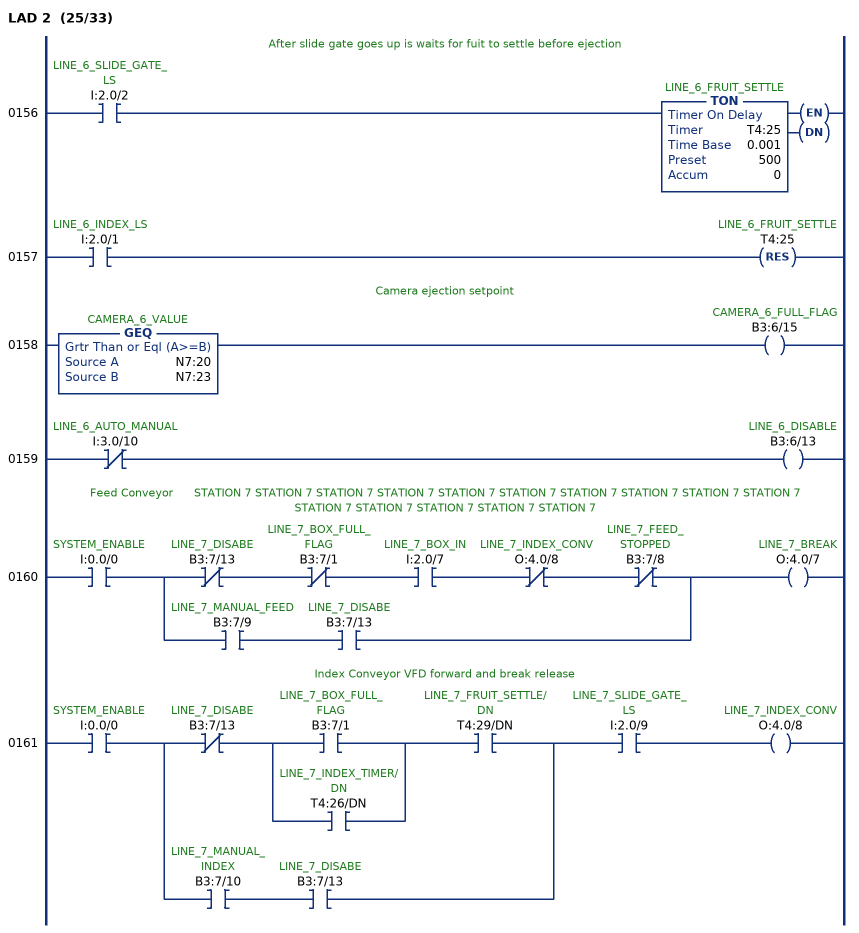
% Rung: 156 %
% After slide gate goes up is waits for fuit to settle before ejection %
SOR XIC I:2.0/2 TON T4:25 0.001 500 0 EOR
%   I:2.0/2  LINE_6_SLIDE_GATE_LS %
%   T4:25  LINE_6_FRUIT_SETTLE %
% Rung: 157 %
SOR XIC I:2.0/1 RES T4:25 EOR
%   I:2.0/1  LINE_6_INDEX_LS %
%   T4:25  LINE_6_FRUIT_SETTLE %
% Rung: 158 %
% Camera ejection setpoint %
SOR GEQ N7:20 N7:23 OTE B3:6/15 EOR
%   N7:20  CAMERA_6_VALUE %
%   N7:23  CAMERA_6_EJECT %
%   B3:6/15  CAMERA_6_FULL_FLAG %
% Rung: 159 %
SOR XIO I:3.0/10 OTE B3:6/13 EOR
%   I:3.0/10  LINE_6_AUTO_MANUAL %
%   B3:6/13  LINE_6_DISABLE %
% Rung: 160 %
% Feed Conveyor      STATION 7 STATION 7 STATION 7 STATION 7 STATION 7 STATION 7 STATION 7 STATION 7 STATION 7 STATION 7 STATION 7 STATION 7 STATION 7 STATION 7 STATION 7 %
SOR XIC I:0.0/0 BST XIO B3:7/13 XIO B3:7/1 XIC I:2.0/7 XIO O:4.0/8 XIO B3:7/8 NXB XIC B3:7/9 XIC B3:7/13 BND OTE O:4.0/7 EOR
%   I:0.0/0  SYSTEM_ENABLE %
%   B3:7/13  LINE_7_DISABE %
%   B3:7/1  LINE_7_BOX_FULL_FLAG %
%   I:2.0/7  LINE_7_BOX_IN %
%   O:4.0/8  LINE_7_INDEX_CONV %
%   B3:7/8  LINE_7_FEED_STOPPED %
%   B3:7/9  LINE_7_MANUAL_FEED %
%   O:4.0/7  LINE_7_BREAK %
% Rung: 161 %
% Index Conveyor VFD forward and break release %
SOR XIC I:0.0/0 BST XIO B3:7/13 BST XIC B3:7/1 NXB XIC T4:26/DN BND XIC T4:29/DN NXB XIC B3:7/10 XIC B3:7/13 BND XIC I:2.0/9 OTE O:4.0/8 EOR
%   I:0.0/0  SYSTEM_ENABLE %
%   B3:7/13  LINE_7_DISABE %
%   B3:7/1  LINE_7_BOX_FULL_FLAG %
%   T4:26  LINE_7_INDEX_TIMER %
%   T4:29  LINE_7_FRUIT_SETTLE %
%   B3:7/10  LINE_7_MANUAL_INDEX %
%   I:2.0/9  LINE_7_SLIDE_GATE_LS %
%   O:4.0/8  LINE_7_INDEX_CONV %

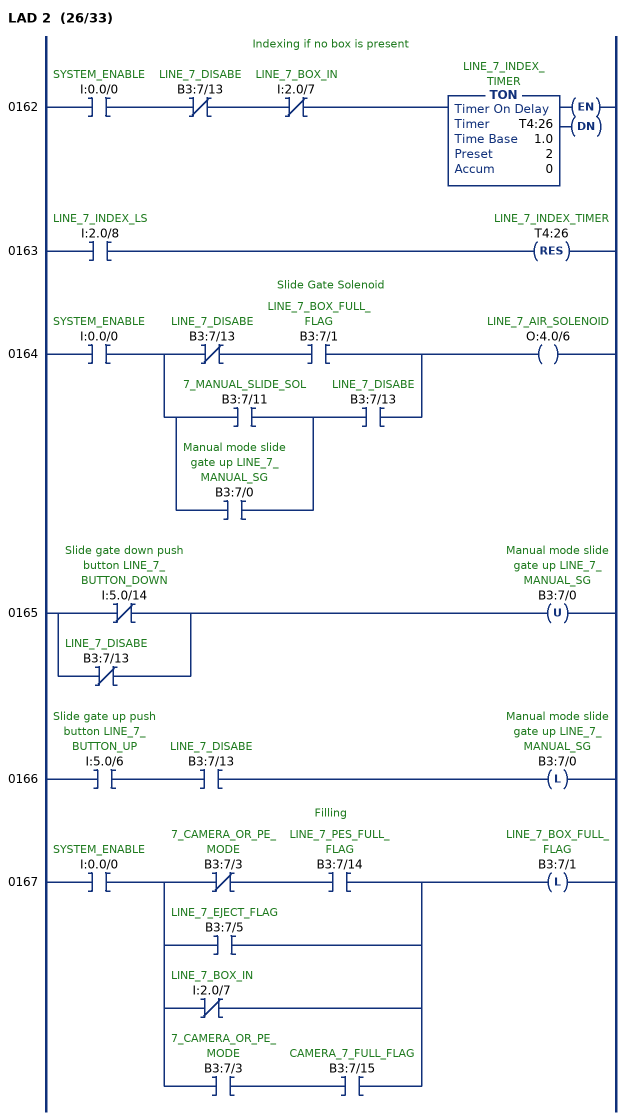
% Rung: 162 %
% Indexing if no box is present %
SOR XIC I:0.0/0 XIO B3:7/13 XIO I:2.0/7 TON T4:26 1.0 2 0 EOR
%   I:0.0/0  SYSTEM_ENABLE %
%   B3:7/13  LINE_7_DISABE %
%   I:2.0/7  LINE_7_BOX_IN %
%   T4:26  LINE_7_INDEX_TIMER %
% Rung: 163 %
SOR XIC I:2.0/8 RES T4:26 EOR
%   I:2.0/8  LINE_7_INDEX_LS %
%   T4:26  LINE_7_INDEX_TIMER %
% Rung: 164 %
% Slide Gate Solenoid %
SOR XIC I:0.0/0 BST XIO B3:7/13 XIC B3:7/1 NXB BST XIC B3:7/11 NXB XIC B3:7/0 BND XIC B3:7/13 BND OTE O:4.0/6 EOR
%   I:0.0/0  SYSTEM_ENABLE %
%   B3:7/13  LINE_7_DISABE %
%   B3:7/1  LINE_7_BOX_FULL_FLAG %
%   B3:7/11  7_MANUAL_SLIDE_SOL %
%   B3:7/0  LINE_7_MANUAL_SG  "Manual mode slide gate up" %
%   O:4.0/6  LINE_7_AIR_SOLENOID %
% Rung: 165 %
SOR BST XIO I:5.0/14 NXB XIO B3:7/13 BND OTU B3:7/0 EOR
%   I:5.0/14  LINE_7_BUTTON_DOWN  "Slide gate down push button" %
%   B3:7/13  LINE_7_DISABE %
%   B3:7/0  LINE_7_MANUAL_SG  "Manual mode slide gate up" %
% Rung: 166 %
SOR XIC I:5.0/6 XIC B3:7/13 OTL B3:7/0 EOR
%   I:5.0/6  LINE_7_BUTTON_UP  "Slide gate up push button" %
%   B3:7/13  LINE_7_DISABE %
%   B3:7/0  LINE_7_MANUAL_SG  "Manual mode slide gate up" %
% Rung: 167 %
% Filling %
SOR XIC I:0.0/0 BST XIO B3:7/3 XIC B3:7/14 NXB BST XIC B3:7/5 NXB BST XIO I:2.0/7 NXB XIC B3:7/3 XIC B3:7/15 BND BND BND OTL B3:7/1 EOR
%   I:0.0/0  SYSTEM_ENABLE %
%   B3:7/3  7_CAMERA_OR_PE_MODE %
%   B3:7/14  LINE_7_PES_FULL_FLAG %
%   B3:7/5  LINE_7_EJECT_FLAG %
%   I:2.0/7  LINE_7_BOX_IN %
%   B3:7/15  CAMERA_7_FULL_FLAG %
%   B3:7/1  LINE_7_BOX_FULL_FLAG %

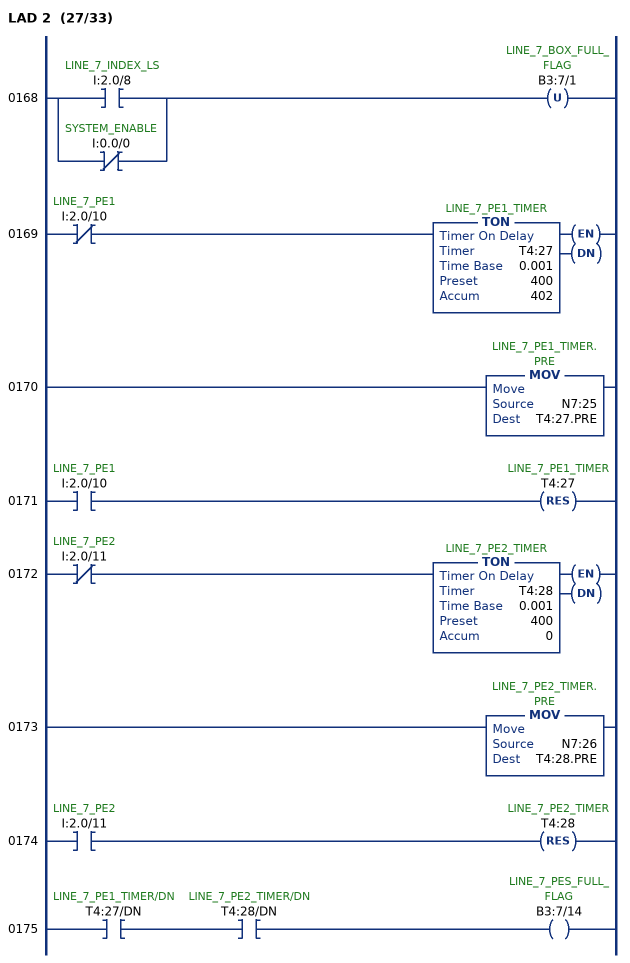
% Rung: 168 %
SOR BST XIC I:2.0/8 NXB XIO I:0.0/0 BND OTU B3:7/1 EOR
%   I:2.0/8  LINE_7_INDEX_LS %
%   I:0.0/0  SYSTEM_ENABLE %
%   B3:7/1  LINE_7_BOX_FULL_FLAG %
% Rung: 169 %
SOR XIO I:2.0/10 TON T4:27 0.001 400 402 EOR
%   I:2.0/10  LINE_7_PE1 %
%   T4:27  LINE_7_PE1_TIMER %
% Rung: 170 %
SOR MOV N7:25 T4:27.PRE EOR
%   N7:25  LINE_7_PE1_TIME_MOV %
%   T4:27  LINE_7_PE1_TIMER %
% Rung: 171 %
SOR XIC I:2.0/10 RES T4:27 EOR
%   I:2.0/10  LINE_7_PE1 %
%   T4:27  LINE_7_PE1_TIMER %
% Rung: 172 %
SOR XIO I:2.0/11 TON T4:28 0.001 400 0 EOR
%   I:2.0/11  LINE_7_PE2 %
%   T4:28  LINE_7_PE2_TIMER %
% Rung: 173 %
SOR MOV N7:26 T4:28.PRE EOR
%   N7:26  LINE_7_PE2_TIME_MOV %
%   T4:28  LINE_7_PE2_TIMER %
% Rung: 174 %
SOR XIC I:2.0/11 RES T4:28 EOR
%   I:2.0/11  LINE_7_PE2 %
%   T4:28  LINE_7_PE2_TIMER %
% Rung: 175 %
SOR XIC T4:27/DN XIC T4:28/DN OTE B3:7/14 EOR
%   T4:27  LINE_7_PE1_TIMER %
%   T4:28  LINE_7_PE2_TIMER %
%   B3:7/14  LINE_7_PES_FULL_FLAG %

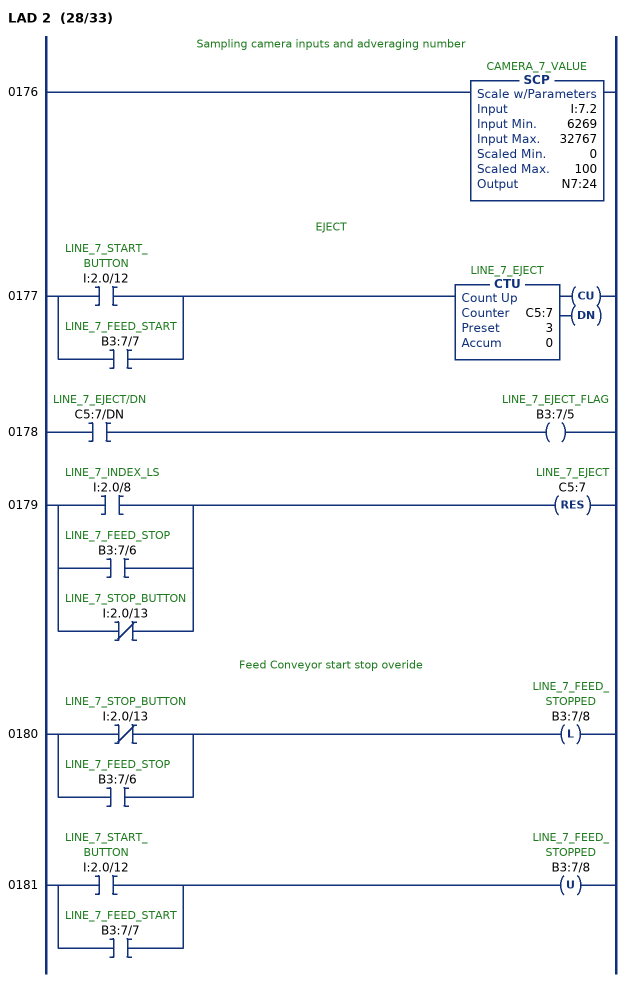
% Rung: 176 %
% Sampling camera inputs and adveraging number %
SOR SCP I:7.2 6269 32767 0 100 N7:24 EOR
%   N7:24  CAMERA_7_VALUE %
% Rung: 177 %
% EJECT %
SOR BST XIC I:2.0/12 NXB XIC B3:7/7 BND CTU C5:7 3 0 EOR
%   I:2.0/12  LINE_7_START_BUTTON %
%   B3:7/7  LINE_7_FEED_START %
%   C5:7  LINE_7_EJECT %
% Rung: 178 %
SOR XIC C5:7/DN OTE B3:7/5 EOR
%   C5:7  LINE_7_EJECT %
%   B3:7/5  LINE_7_EJECT_FLAG %
% Rung: 179 %
SOR BST XIC I:2.0/8 NXB BST XIC B3:7/6 NXB XIO I:2.0/13 BND BND RES C5:7 EOR
%   I:2.0/8  LINE_7_INDEX_LS %
%   B3:7/6  LINE_7_FEED_STOP %
%   I:2.0/13  LINE_7_STOP_BUTTON %
%   C5:7  LINE_7_EJECT %
% Rung: 180 %
% Feed Conveyor start stop overide %
SOR BST XIO I:2.0/13 NXB XIC B3:7/6 BND OTL B3:7/8 EOR
%   I:2.0/13  LINE_7_STOP_BUTTON %
%   B3:7/6  LINE_7_FEED_STOP %
%   B3:7/8  LINE_7_FEED_STOPPED %
% Rung: 181 %
SOR BST XIC I:2.0/12 NXB XIC B3:7/7 BND OTU B3:7/8 EOR
%   I:2.0/12  LINE_7_START_BUTTON %
%   B3:7/7  LINE_7_FEED_START %
%   B3:7/8  LINE_7_FEED_STOPPED %

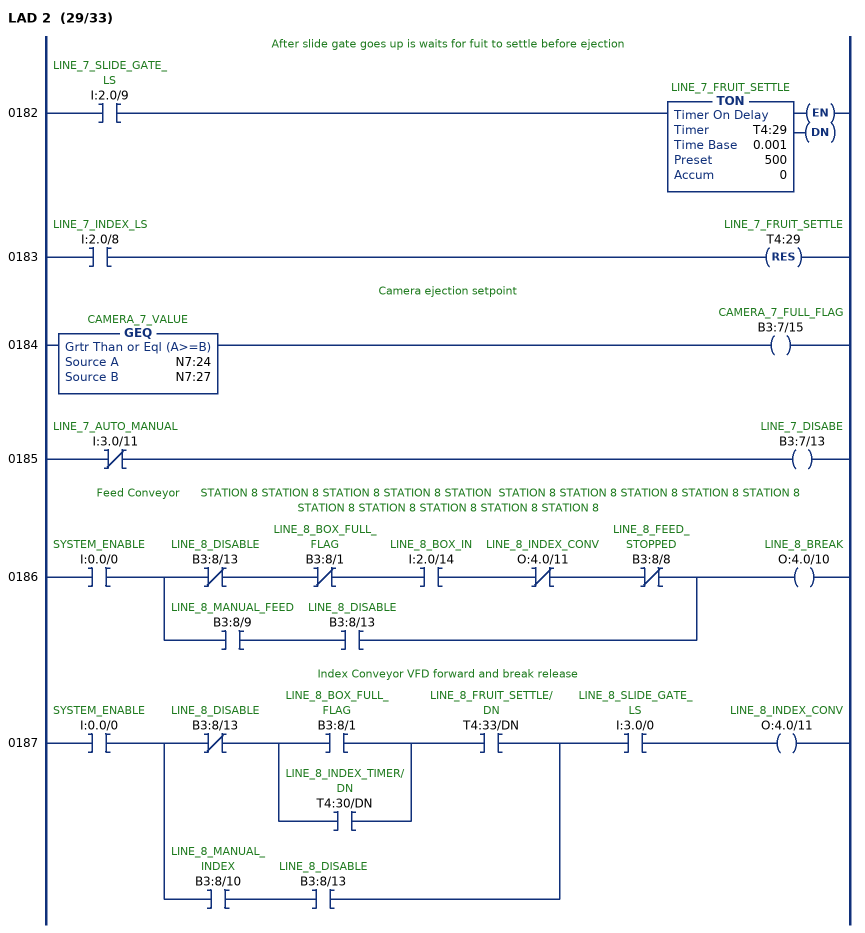
% Rung: 182 %
% After slide gate goes up is waits for fuit to settle before ejection %
SOR XIC I:2.0/9 TON T4:29 0.001 500 0 EOR
%   I:2.0/9  LINE_7_SLIDE_GATE_LS %
%   T4:29  LINE_7_FRUIT_SETTLE %
% Rung: 183 %
SOR XIC I:2.0/8 RES T4:29 EOR
%   I:2.0/8  LINE_7_INDEX_LS %
%   T4:29  LINE_7_FRUIT_SETTLE %
% Rung: 184 %
% Camera ejection setpoint %
SOR GEQ N7:24 N7:27 OTE B3:7/15 EOR
%   N7:24  CAMERA_7_VALUE %
%   N7:27  CAMERA_7_EJECT %
%   B3:7/15  CAMERA_7_FULL_FLAG %
% Rung: 185 %
SOR XIO I:3.0/11 OTE B3:7/13 EOR
%   I:3.0/11  LINE_7_AUTO_MANUAL %
%   B3:7/13  LINE_7_DISABE %
% Rung: 186 %
% Feed Conveyor      STATION 8 STATION 8 STATION 8 STATION 8 STATION  STATION 8 STATION 8 STATION 8 STATION 8 STATION 8 STATION 8 STATION 8 STATION 8 STATION 8 STATION 8 %
SOR XIC I:0.0/0 BST XIO B3:8/13 XIO B3:8/1 XIC I:2.0/14 XIO O:4.0/11 XIO B3:8/8 NXB XIC B3:8/9 XIC B3:8/13 BND OTE O:4.0/10 EOR
%   I:0.0/0  SYSTEM_ENABLE %
%   B3:8/13  LINE_8_DISABLE %
%   B3:8/1  LINE_8_BOX_FULL_FLAG %
%   I:2.0/14  LINE_8_BOX_IN %
%   O:4.0/11  LINE_8_INDEX_CONV %
%   B3:8/8  LINE_8_FEED_STOPPED %
%   B3:8/9  LINE_8_MANUAL_FEED %
%   O:4.0/10  LINE_8_BREAK %
% Rung: 187 %
% Index Conveyor VFD forward and break release %
SOR XIC I:0.0/0 BST XIO B3:8/13 BST XIC B3:8/1 NXB XIC T4:30/DN BND XIC T4:33/DN NXB XIC B3:8/10 XIC B3:8/13 BND XIC I:3.0/0 OTE O:4.0/11 EOR
%   I:0.0/0  SYSTEM_ENABLE %
%   B3:8/13  LINE_8_DISABLE %
%   B3:8/1  LINE_8_BOX_FULL_FLAG %
%   T4:30  LINE_8_INDEX_TIMER %
%   T4:33  LINE_8_FRUIT_SETTLE %
%   B3:8/10  LINE_8_MANUAL_INDEX %
%   I:3.0/0  LINE_8_SLIDE_GATE_LS %
%   O:4.0/11  LINE_8_INDEX_CONV %

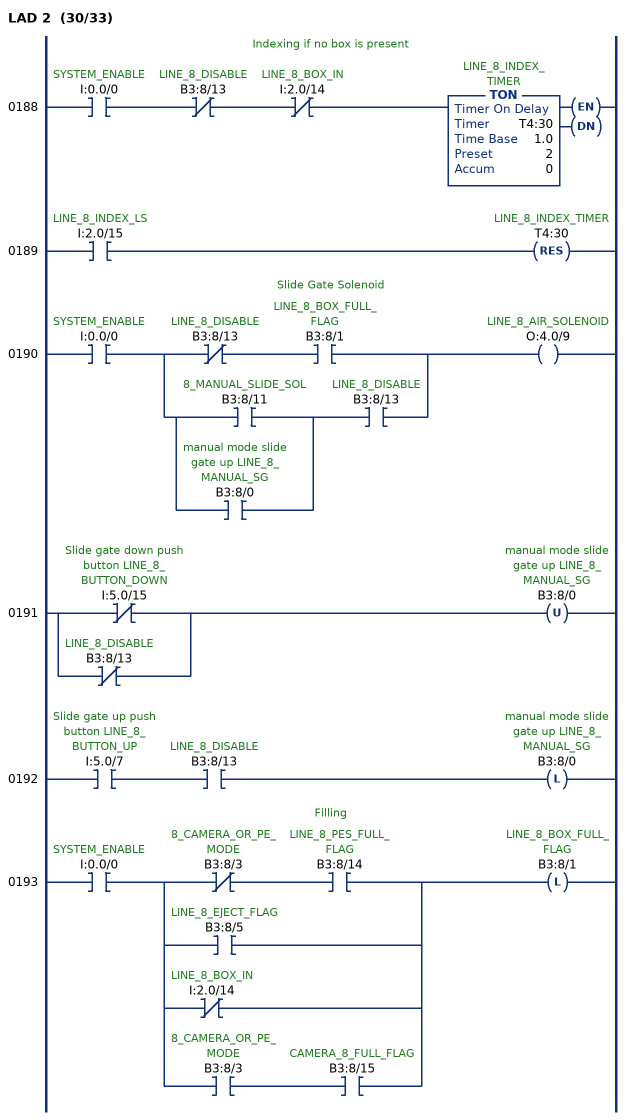
% Rung: 188 %
% Indexing if no box is present %
SOR XIC I:0.0/0 XIO B3:8/13 XIO I:2.0/14 TON T4:30 1.0 2 0 EOR
%   I:0.0/0  SYSTEM_ENABLE %
%   B3:8/13  LINE_8_DISABLE %
%   I:2.0/14  LINE_8_BOX_IN %
%   T4:30  LINE_8_INDEX_TIMER %
% Rung: 189 %
SOR XIC I:2.0/15 RES T4:30 EOR
%   I:2.0/15  LINE_8_INDEX_LS %
%   T4:30  LINE_8_INDEX_TIMER %
% Rung: 190 %
% Slide Gate Solenoid %
SOR XIC I:0.0/0 BST XIO B3:8/13 XIC B3:8/1 NXB BST XIC B3:8/11 NXB XIC B3:8/0 BND XIC B3:8/13 BND OTE O:4.0/9 EOR
%   I:0.0/0  SYSTEM_ENABLE %
%   B3:8/13  LINE_8_DISABLE %
%   B3:8/1  LINE_8_BOX_FULL_FLAG %
%   B3:8/11  8_MANUAL_SLIDE_SOL %
%   B3:8/0  LINE_8_MANUAL_SG  "manual mode slide gate up" %
%   O:4.0/9  LINE_8_AIR_SOLENOID %
% Rung: 191 %
SOR BST XIO I:5.0/15 NXB XIO B3:8/13 BND OTU B3:8/0 EOR
%   I:5.0/15  LINE_8_BUTTON_DOWN  "Slide gate down push button" %
%   B3:8/13  LINE_8_DISABLE %
%   B3:8/0  LINE_8_MANUAL_SG  "manual mode slide gate up" %
% Rung: 192 %
SOR XIC I:5.0/7 XIC B3:8/13 OTL B3:8/0 EOR
%   I:5.0/7  LINE_8_BUTTON_UP  "Slide gate up push button" %
%   B3:8/13  LINE_8_DISABLE %
%   B3:8/0  LINE_8_MANUAL_SG  "manual mode slide gate up" %
% Rung: 193 %
% Filling %
SOR XIC I:0.0/0 BST XIO B3:8/3 XIC B3:8/14 NXB BST XIC B3:8/5 NXB BST XIO I:2.0/14 NXB XIC B3:8/3 XIC B3:8/15 BND BND BND OTL B3:8/1 EOR
%   I:0.0/0  SYSTEM_ENABLE %
%   B3:8/3  8_CAMERA_OR_PE_MODE %
%   B3:8/14  LINE_8_PES_FULL_FLAG %
%   B3:8/5  LINE_8_EJECT_FLAG %
%   I:2.0/14  LINE_8_BOX_IN %
%   B3:8/15  CAMERA_8_FULL_FLAG %
%   B3:8/1  LINE_8_BOX_FULL_FLAG %

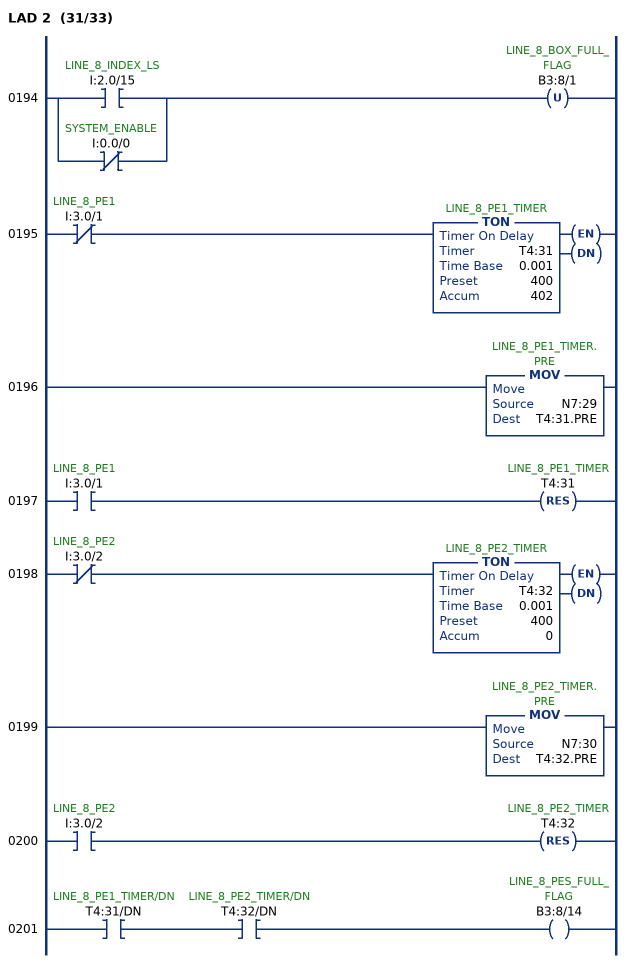
% Rung: 194 %
SOR BST XIC I:2.0/15 NXB XIO I:0.0/0 BND OTU B3:8/1 EOR
%   I:2.0/15  LINE_8_INDEX_LS %
%   I:0.0/0  SYSTEM_ENABLE %
%   B3:8/1  LINE_8_BOX_FULL_FLAG %
% Rung: 195 %
SOR XIO I:3.0/1 TON T4:31 0.001 400 402 EOR
%   I:3.0/1  LINE_8_PE1 %
%   T4:31  LINE_8_PE1_TIMER %
% Rung: 196 %
SOR MOV N7:29 T4:31.PRE EOR
%   N7:29  LINE_8_PE1_TIME_MOV %
%   T4:31  LINE_8_PE1_TIMER %
% Rung: 197 %
SOR XIC I:3.0/1 RES T4:31 EOR
%   I:3.0/1  LINE_8_PE1 %
%   T4:31  LINE_8_PE1_TIMER %
% Rung: 198 %
SOR XIO I:3.0/2 TON T4:32 0.001 400 0 EOR
%   I:3.0/2  LINE_8_PE2 %
%   T4:32  LINE_8_PE2_TIMER %
% Rung: 199 %
SOR MOV N7:30 T4:32.PRE EOR
%   N7:30  LINE_8_PE2_TIME_MOV %
%   T4:32  LINE_8_PE2_TIMER %
% Rung: 200 %
SOR XIC I:3.0/2 RES T4:32 EOR
%   I:3.0/2  LINE_8_PE2 %
%   T4:32  LINE_8_PE2_TIMER %
% Rung: 201 %
SOR XIC T4:31/DN XIC T4:32/DN OTE B3:8/14 EOR
%   T4:31  LINE_8_PE1_TIMER %
%   T4:32  LINE_8_PE2_TIMER %
%   B3:8/14  LINE_8_PES_FULL_FLAG %

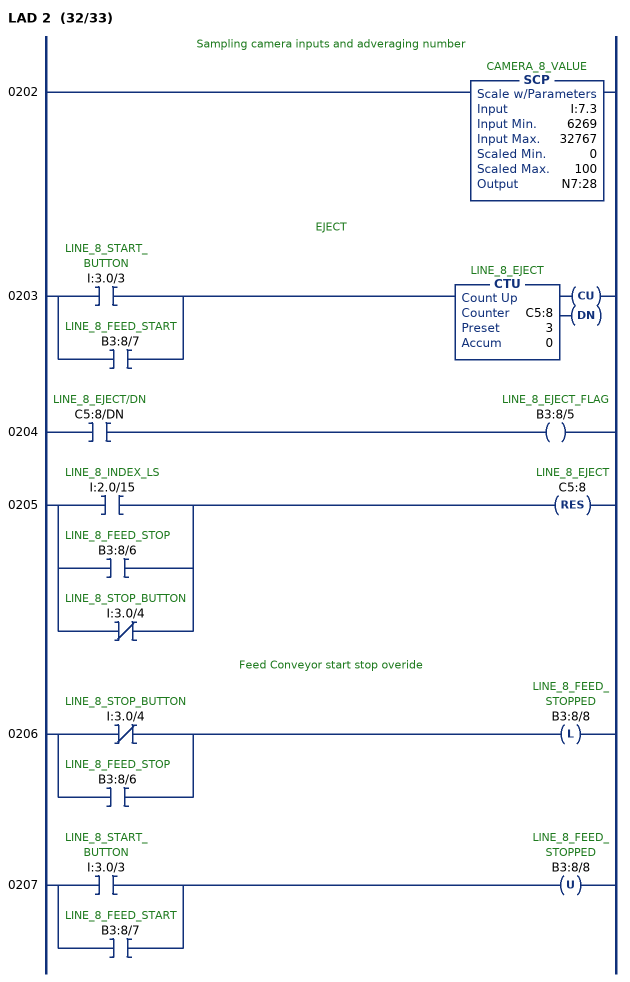
% Rung: 202 %
% Sampling camera inputs and adveraging number %
SOR SCP I:7.3 6269 32767 0 100 N7:28 EOR
%   N7:28  CAMERA_8_VALUE %
% Rung: 203 %
% EJECT %
SOR BST XIC I:3.0/3 NXB XIC B3:8/7 BND CTU C5:8 3 0 EOR
%   I:3.0/3  LINE_8_START_BUTTON %
%   B3:8/7  LINE_8_FEED_START %
%   C5:8  LINE_8_EJECT %
% Rung: 204 %
SOR XIC C5:8/DN OTE B3:8/5 EOR
%   C5:8  LINE_8_EJECT %
%   B3:8/5  LINE_8_EJECT_FLAG %
% Rung: 205 %
SOR BST XIC I:2.0/15 NXB BST XIC B3:8/6 NXB XIO I:3.0/4 BND BND RES C5:8 EOR
%   I:2.0/15  LINE_8_INDEX_LS %
%   B3:8/6  LINE_8_FEED_STOP %
%   I:3.0/4  LINE_8_STOP_BUTTON %
%   C5:8  LINE_8_EJECT %
% Rung: 206 %
% Feed Conveyor start stop overide %
SOR BST XIO I:3.0/4 NXB XIC B3:8/6 BND OTL B3:8/8 EOR
%   I:3.0/4  LINE_8_STOP_BUTTON %
%   B3:8/6  LINE_8_FEED_STOP %
%   B3:8/8  LINE_8_FEED_STOPPED %
% Rung: 207 %
SOR BST XIC I:3.0/3 NXB XIC B3:8/7 BND OTU B3:8/8 EOR
%   I:3.0/3  LINE_8_START_BUTTON %
%   B3:8/7  LINE_8_FEED_START %
%   B3:8/8  LINE_8_FEED_STOPPED %

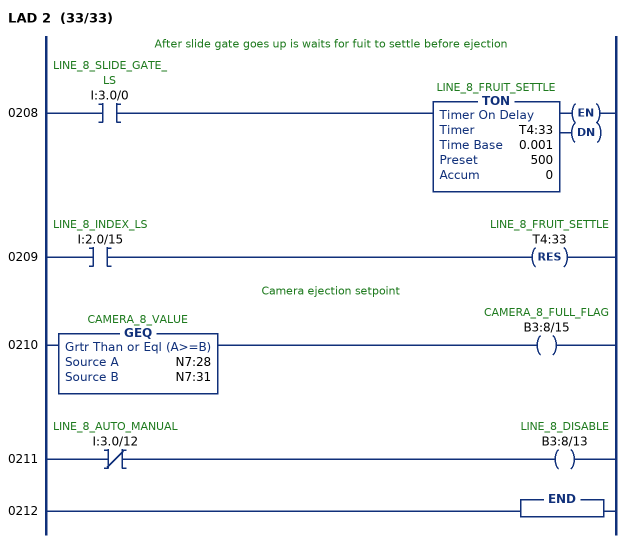
% Rung: 208 %
% After slide gate goes up is waits for fuit to settle before ejection %
SOR XIC I:3.0/0 TON T4:33 0.001 500 0 EOR
%   I:3.0/0  LINE_8_SLIDE_GATE_LS %
%   T4:33  LINE_8_FRUIT_SETTLE %
% Rung: 209 %
SOR XIC I:2.0/15 RES T4:33 EOR
%   I:2.0/15  LINE_8_INDEX_LS %
%   T4:33  LINE_8_FRUIT_SETTLE %
% Rung: 210 %
% Camera ejection setpoint %
SOR GEQ N7:28 N7:31 OTE B3:8/15 EOR
%   N7:28  CAMERA_8_VALUE %
%   N7:31  CAMERA_8_EJECT %
%   B3:8/15  CAMERA_8_FULL_FLAG %
% Rung: 211 %
SOR XIO I:3.0/12 OTE B3:8/13 EOR
%   I:3.0/12  LINE_8_AUTO_MANUAL %
%   B3:8/13  LINE_8_DISABLE %
% Rung: 212 %
SOR END EOR

OTHER DOCUMENTED ADDRESSES
  B3:0/4  1_BOX_FULL_UNLATCH  "Box Full Unlatch"
  B3:2/4  2_BOX_FULL_UNLATCH
  B3:3/4  3_BOX_FULL_UNLATCH
  B3:4/4  4_BOX_FULL_UNLATCH
  B3:5/4  5_BOX_FULL_UNLATCH
  B3:6/4  6_BOX_FULL_UNLATCH
  B3:7/4  7_BOX_FULL_UNLATCH
  B3:8/4  8_BOX_FULL_UNLATCH
  C5:0.ACC  "Counter"
  C5:0/DN  COUNT_DONE
  I:6.0/0  CAMERA_1  "Camera 1 4-20 input"
  I:7.0/0  CAMERA_5  "Camera 1 4-20 input"

REVISION NOTES
  0: Simplified

DATA TABLE (non-zero values as saved)
DATA B3
% B3:0 % 0X0008 0X000B 0X0008 0X0008 0X0808 0X0008 0X0008 0X0008 0X0008 0X0001
DATA T4
% .PRE .ACC %
% T4:0 % 2 0
% T4:1 % 400 0
% T4:2 % 1 0
% T4:3 % 1 0
% T4:4 % 400 401
% T4:5 % 500 0
% T4:6 % 2 0
% T4:7 % 400 0
% T4:8 % 400 0
% T4:9 % 500 0
% T4:10 % 2 0
% T4:11 % 400 0
% T4:12 % 400 0
% T4:13 % 500 0
% T4:14 % 2 0
% T4:15 % 200 0
% T4:16 % 200 0
% T4:17 % 500 0
% T4:18 % 2 0
% T4:19 % 400 0
% T4:20 % 400 0
% T4:21 % 500 0
% T4:22 % 2 0
% T4:23 % 400 0
% T4:24 % 400 0
% T4:25 % 500 0
% T4:26 % 2 0
% T4:27 % 400 402
% T4:28 % 400 0
% T4:29 % 500 0
% T4:30 % 2 0
% T4:31 % 400 402
% T4:32 % 400 0
% T4:33 % 500 0
DATA C5
% .PRE .ACC %
% C5:0 % 6 1
% C5:1 % 3 0
% C5:2 % 3 0
% C5:3 % 3 0
% C5:4 % 3 0
% C5:5 % 3 0
% C5:6 % 3 1
% C5:7 % 3 0
% C5:8 % 3 0
DATA N7
% N7:0 % 9 400 400 27 4 400 400 20 21 400
% N7:10 % 400 27 -10 200 200 27 -11 400 400 24
% N7:20 % 12 400 400 35 -12 400 400 35 15 400
% N7:30 % 400 35 400
DATA F8
% F8:0 % 0 22161 86.55965
